Staubli VAL3: buildList.pgx

program buildList()
  local num l_nSize
  local string l_sEvent
  local num i
  local string l_sEmpty
begin
  // INIT the list
  call use:stringCopy(l_sEmpty,sList)
  // Build the list

end
